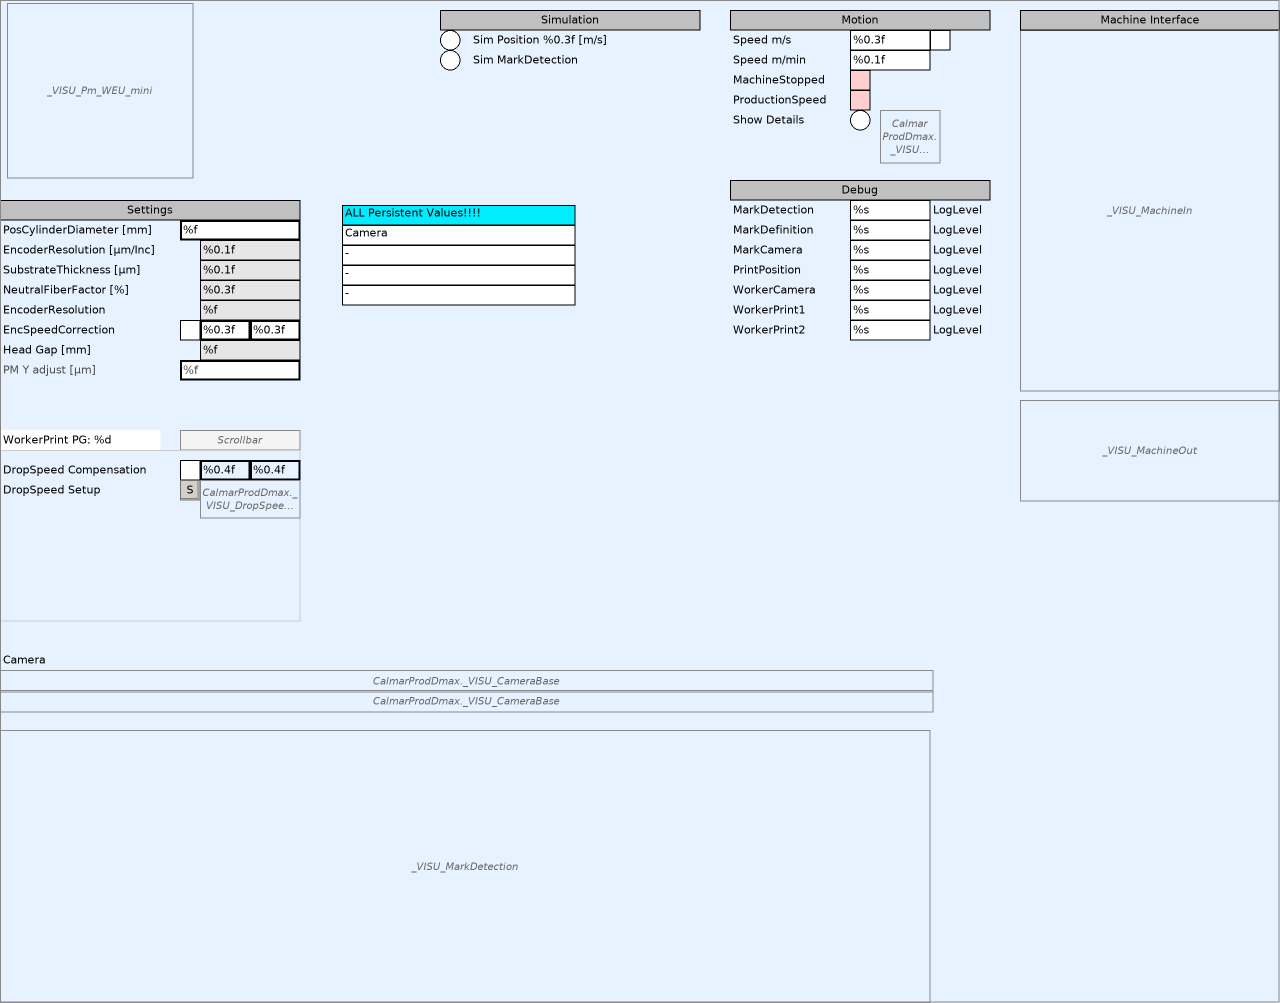
VISUALIZATION _VISU_Pm_WEU  // 1280x1003
VAR_IN_OUT
  mInst : FB_PrintModule_WEU;
END_VAR
    Rectangle (730,30 120x20), "Speed m/s"
    Rectangle (850,30 80x20), "%0.3f", text variable: mInst.fSpeed
    RoundedRectangle (850,70 20x20), colour toggle: mInst.bMoving
    Rectangle (730,70 110x20), "MachineStopped"
    RoundedRectangle (850,90 20x20), colour toggle: mInst.bProductionSpeedReached
    Rectangle (730,90 110x20), "ProductionSpeed"
    Rectangle (730,50 120x20), "Speed m/min"
    Rectangle (850,50 80x20), "%0.1f", text variable: mInst.fSpeedMpMin
    Rectangle (0,220 180x20), "PosCylinderDiameter [mm]"
    Rectangle (0,240 180x20), "EncoderResolution [µm/Inc]"
    Rectangle (200,240 100x20), "%0.1f", text variable: mInst.fC_EncoderImpU
    Rectangle (180,220 120x20), "%f", text variable: mInst._fEncoderCylinderDiameter
        OnMouseClick: write the text variable via Default
    Rectangle (0,260 180x20), "SubstrateThickness [µm]"
    Rectangle (200,260 100x20), "%0.1f", text variable: mInst._pModuleMachineState^.fSubstrateThickness * 1_000_000
    Rectangle (0,360 180x20), "PM Y adjust [µm]"
    Rectangle (180,360 120x20), "%f", text variable: mInst._fPrintModuleAdjustY
        OnMouseClick: write the text variable via VisuDialogs.Numpad, min PRG_PRINT.sC_Config_P.lL_PU_GENERALSHIFT_Y_SET_MIN, max PRG_PRINT.sC_Config_P.lL_PU_GENERALSHIFT_Y_SET_MAX
    Rectangle (0,340 180x20), "Head Gap [mm]"
    Rectangle (200,340 100x20), "%f", text variable: mInst._pAdsSa^.sI_HeadGap.fI_Val
        OnMouseClick: write the text variable via Default
    RoundedRectangle (930,30 20x20), tooltip "Exeeds max. speed=%f", colour toggle: mInst._pModuleMachineFeedback^.bSpeedExeeded
        p4168582468: mInst._pModuleMachineFeedback^.fMaxSpeed
    Frame (1020,400 260x101)
        shows _VISU_MachineOut(ref := mInst._pModuleMachineFeedback^)
    Frame (1020,30 260x361)
        shows _VISU_MachineIn(ref := mInst._pModuleMachineState^)
    Rectangle (1020,10 260x20), "Machine Interface"
    Rectangle (730,10 260x20), "Motion"
    Frame (0,670 933x22)
        shows CalmarProdDmax._VISU_CameraBase(m_Inst := mInst.fbMarkCameraWeu)
    Frame (0,690 933x22)
        shows CalmarProdDmax._VISU_CameraBase(m_Inst := mInst.fbNoCamera)
    Rectangle (0,650 120x20), "Camera"
    Rectangle (440,10 260x20), "Simulation"
    Ellipse (440,30 20x20), tooltip "Sim position"
        toggle mInst.fbPrintPosition._bSim
    Rectangle (470,30 200x20), "Sim Position %0.3f [m/s]", text variable: mInst.fbPrintPosition.fbPositionMaster.fSimSpeed
        OnMouseClick: write the text variable via Default
    Frame (7,3 186x175)
        shows _VISU_Pm_WEU_mini(mInst := mInst)
    Rectangle (730,110 110x20), "Show Details"
    Ellipse (850,110 20x20)
        toggle mInst.fbView.bShowPositionDetail
    Rectangle (0,200 300x20), "Settings"
    RoundedRectangle (342,225 233x20), "Camera"
    RoundedRectangle (342,245 233x20), "-"
    RoundedRectangle (342,265 233x20), "-"
    RoundedRectangle (342,285 233x20), "-"
    RoundedRectangle (342,205 233x20), "ALL Persistent Values!!!!"
    Rectangle (250,320 50x20), "%0.3f", tooltip "Encoder speed compensation reference speed", text variable: mInst.fbPrintPosition._fSpeedCompRefSpeed
        OnMouseClick: write the text variable via Default
    Rectangle (200,320 50x20), "%0.3f", tooltip "Encoder speed compensation factor", text variable: mInst.fbPrintPosition._fSpeedCompFactor
        OnMouseClick: write the text variable via Default
    RoundedRectangle (180,320 20x20)
        toggle mInst.fbPrintPosition._bEnSpeedComp
    Rectangle (0,320 180x20), "EncSpeedCorrection"
    Rectangle (0,300 180x20), "EncoderResolution"
    Rectangle (200,300 100x20), "%f", text variable: mInst.fbPrintPosition._fEncoderResolution
    Rectangle (0,280 180x20), "NeutralFiberFactor [%]"
    Rectangle (200,280 100x20), "%0.3f", text variable: mInst._pModuleMachineState^.fNeutralFibreFactor
    Scrollbar (180,430 120x20)
        p2245068023: GVL_WEU.nC_WorkerPrintPerPm
        p1057716461: mInst.fbView.nSelWorkerPrint
    Rectangle (0,430 160x20), "WorkerPrint PG: %d", text variable: mInst.fbView.nSelWorkerPrint
    Rectangle (0,450 300x171)
    Rectangle (0,460 180x20), "DropSpeed Compensation"
    Rectangle (200,460 50x20), "%0.4f", tooltip "DropSpeed [m/s]", text variable: mInst.fbWorkerPrint[mInst.fbView.nSelWorkerPrint].fbDropSpeedComp.fDropSpeed
        OnMouseClick: write the text variable via Default
    Rectangle (250,460 50x20), "%0.4f", tooltip "Dead/Add Time [ms]", text variable: mInst.fbWorkerPrint[mInst.fbView.nSelWorkerPrint].fbDropSpeedComp.fDropSpeedDeadTime
        OnMouseClick: write the text variable via Default
    RoundedRectangle (180,460 20x20), tooltip "Enabled compensation", input disabled if: TRUE
        toggle mInst.fbWorkerPrint[mInst.fbView.nSelWorkerPrint].fbDropSpeedComp._bEnable p2164770859=TRUE
    Button (180,480 20x20), "S", tooltip "Setup"
        toggle minst.fbView.bShowDropSpeedSetup
    Rectangle (0,480 180x20), "DropSpeed Setup"
    Frame (0,730 930x273)
        shows _VISU_MarkDetection(mInst := mInst.fbMarkDetection)
    Ellipse (440,50 20x20), tooltip "Sim position"
        toggle mInst.fbMarkDetection.bSimEnable
    Rectangle (470,50 200x20), "Sim MarkDetection"
    Rectangle (730,180 260x20), "Debug"
    Rectangle (730,200 120x20), "MarkDetection"
    Rectangle (930,200 60x20), "LogLevel"
        OnMouseClick: write the text variable via Default
    Rectangle (850,200 80x20), "%s", text variable: mInst.fbMarkDetection._loglevel
        OnMouseClick: write the text variable via Default
    Rectangle (730,220 120x20), "MarkDefinition"
    Rectangle (930,220 60x20), "LogLevel"
        OnMouseClick: write the text variable via Default
    Rectangle (850,220 80x20), "%s", text variable: mInst.fbMarkDefinition._loglevel
        OnMouseClick: write the text variable via Default
    Rectangle (730,240 120x20), "MarkCamera"
    Rectangle (930,240 60x20), "LogLevel"
        OnMouseClick: write the text variable via Default
    Rectangle (850,240 80x20), "%s", text variable: mInst.fbMarkCameraWeu._loglevel
        OnMouseClick: write the text variable via Default
    Rectangle (930,260 60x20), "LogLevel"
        OnMouseClick: write the text variable via Default
    Rectangle (730,260 120x20), "PrintPosition"
    Rectangle (850,260 80x20), "%s", text variable: mInst.fbPrintPosition._loglevel
        OnMouseClick: write the text variable via Default
    Rectangle (730,280 120x20), "WorkerCamera"
    Rectangle (930,280 60x20), "LogLevel"
        OnMouseClick: write the text variable via Default
    Rectangle (850,280 80x20), "%s", text variable: mInst.fbWorkerCamera._loglevel
        OnMouseClick: write the text variable via Default
    Rectangle (930,300 60x20), "LogLevel"
        OnMouseClick: write the text variable via Default
    Rectangle (730,300 120x20), "WorkerPrint1"
    Rectangle (850,300 80x20), "%s", text variable: mInst.fbWorkerPrint[1]._loglevel
        OnMouseClick: write the text variable via Default
    Rectangle (930,320 60x20), "LogLevel"
        OnMouseClick: write the text variable via Default
    Rectangle (730,320 120x20), "WorkerPrint2"
    Rectangle (850,320 80x20), "%s", text variable: mInst.fbWorkerPrint[2]._loglevel
        OnMouseClick: write the text variable via Default
    Frame (200,480 100x38), invisible if: NOT minst.fbView.bShowDropSpeedSetup
        shows CalmarProdDmax._VISU_DropSpeedComp_Setup(mInst := mInst.fbWorkerPrint[mInst.fbView.nSelWorkerPrint].fbDropSpeedComp)
    Frame (880,110 60x53), invisible if: NOT mInst.fbView.bShowPositionDetail
        shows CalmarProdDmax._VISU_PrintPositionDmax(m_Inst := mInst.fbPrintPosition)
END_VISUALIZATION

(* stored: Version 1.1.0.1, ProductVersion 3.1.4024.11
   Visu _VISU_Pm_WEU: Id {1c33c1d3-4cba-4983-923f-6027f0964b30} *)
